(*
SPDX-FileCopyrightText: © 2026 Oleksandr Tiutyk <trofimich@gmail.com>
SPDX-License-Identifier: MIT
License: https://opensource.org/license/mit
*)

INTERFACE IArgumentNotSpecifiedException EXTENDS IGeneralException

METHOD Throw
VAR_INPUT
	sourceNamespaceName : STRING;
	sourceClassName : STRING;
	sourcePOUName : STRING;
	sourcePosition : STRING;
	argumentName : STRING;
END_VAR
END_METHOD

END_INTERFACE

(* stored: Version 1.1.0.1
   Itf IArgumentNotSpecifiedException: Id {8d1dcd2c-ca51-4f93-8b0f-4c12ec4ce6a4}
   Method Throw: Id {170f19d7-15b2-43f5-807c-aef9f4d86d53} *)
